FUNCTION CountDefects : INT
VAR_INPUT
	aRefArray : REFERENCE TO ARRAY[1..20] OF REAL;
END_VAR
VAR
	
	nIterator: INT;
END_VAR

FOR nIterator := 1 TO 20 DO
	IF aRefArray[nIterator] < 50 THEN
		CountDefects := CountDefects + 1;
	END_IF
	IF aRefArray[nIterator] > 500 THEN
		CountDefects := CountDefects + 1;
	END_IF
END_FOR

END_FUNCTION

(* stored: Version 1.1.0.1, ProductVersion 3.1.4024.16
   POU CountDefects: Id {4c35b219-d7dc-4f39-b38f-a6c35a698867}, SpecialFunc None *)
